// TIA Portal V19 export
FUNCTION "CallDiagnostic" : Void   // FC16, LAD
TITLE = Diagnostics / Diagnose
AUTHOR : Siemens Digital Industries
// Call of diagnostic blocks / Aufruf: Diagnose
// stored: IsIECCheckEnabled true, SetENOAutomatically true
   // Ret_Val : Ret_Val
BEGIN

REGION Network 1: Call Profinet Devices Diagnostics
   // For diagnostics of all profinet devices of this PLC
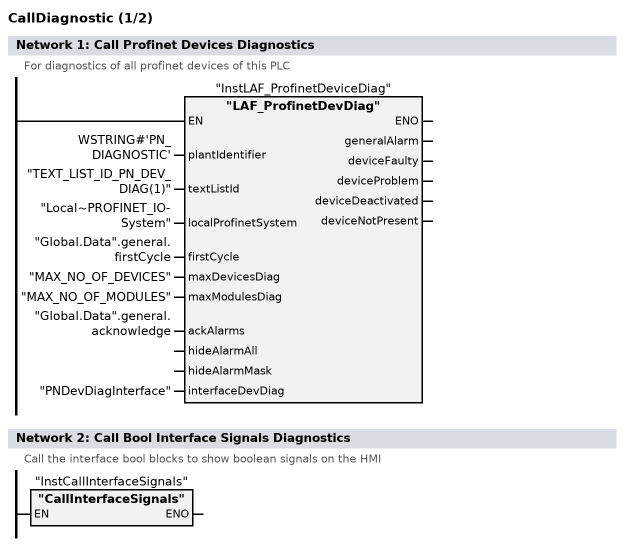
   RUNG wire#powerrail
      "InstLAF_ProfinetDeviceDiag"(plantIdentifier := WSTRING#'PN_DIAGNOSTIC', textListId := "TEXT_LIST_ID_PN_DEV_DIAG(1)", localProfinetSystem := "Local~PROFINET_IO-System", firstCycle := "Global.Data".general.firstCycle, maxDevicesDiag := "MAX_NO_OF_DEVICES", maxModulesDiag := "MAX_NO_OF_MODULES", ackAlarms := "Global.Data".general.acknowledge, hideAlarmAll :=, hideAlarmMask :=, interfaceDevDiag := "PNDevDiagInterface", generalAlarm =>, deviceFaulty =>, deviceProblem =>, deviceDeactivated =>, deviceNotPresent =>)
   END_RUNG
   // the same network as SCL:
   "InstLAF_ProfinetDeviceDiag"(plantIdentifier := WSTRING#'PN_DIAGNOSTIC',   // "LAF_ProfinetDevDiag"
                           textListId := "TEXT_LIST_ID_PN_DEV_DIAG(1)",
                           localProfinetSystem := "Local~PROFINET_IO-System",
                           firstCycle := "Global.Data".general.firstCycle,
                           maxDevicesDiag := "MAX_NO_OF_DEVICES",
                           maxModulesDiag := "MAX_NO_OF_MODULES",
                           ackAlarms := "Global.Data".general.acknowledge,
                           interfaceDevDiag := "PNDevDiagInterface");
END_REGION

REGION Network 2: Call Bool Interface Signals Diagnostics
   // Call the interface bool blocks to show boolean signals on the HMI
   RUNG wire#powerrail
      "InstCallInterfaceSignals"()
   END_RUNG
   // the same network as SCL:
   "InstCallInterfaceSignals"();   // "CallInterfaceSignals"
END_REGION

REGION Network 3: Call Drives Diagnostics
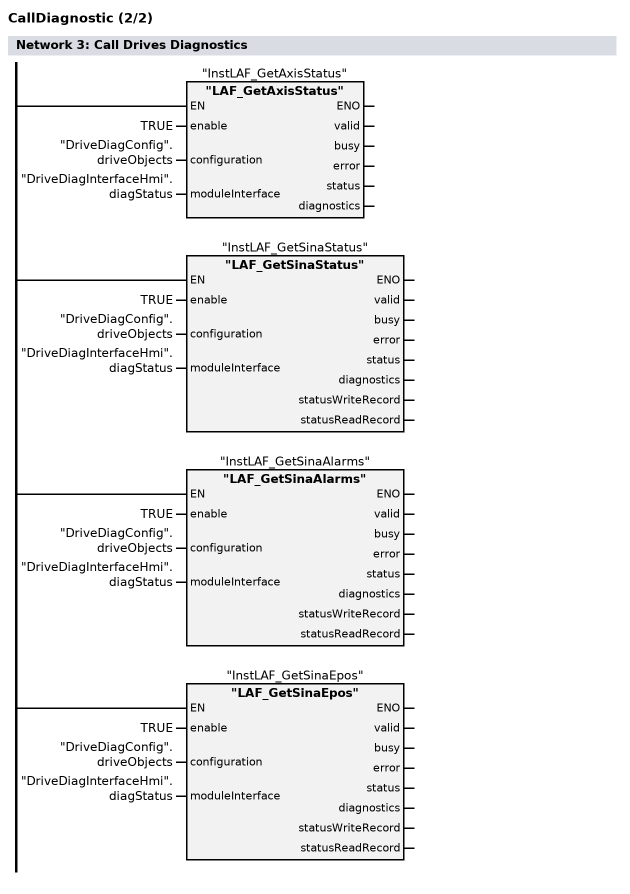
   RUNG wire#powerrail
      "InstLAF_GetAxisStatus"(enable := TRUE, configuration := "DriveDiagConfig".driveObjects, moduleInterface := "DriveDiagInterfaceHmi".diagStatus, valid =>, busy =>, error =>, status =>, diagnostics =>)
   END_RUNG
   RUNG wire#powerrail
      "InstLAF_GetSinaStatus"(enable := TRUE, configuration := "DriveDiagConfig".driveObjects, moduleInterface := "DriveDiagInterfaceHmi".diagStatus, valid =>, busy =>, error =>, status =>, diagnostics =>, statusWriteRecord =>, statusReadRecord =>)
   END_RUNG
   RUNG wire#powerrail
      "InstLAF_GetSinaAlarms"(enable := TRUE, configuration := "DriveDiagConfig".driveObjects, moduleInterface := "DriveDiagInterfaceHmi".diagStatus, valid =>, busy =>, error =>, status =>, diagnostics =>, statusWriteRecord =>, statusReadRecord =>)
   END_RUNG
   RUNG wire#powerrail
      "InstLAF_GetSinaEpos"(enable := TRUE, configuration := "DriveDiagConfig".driveObjects, moduleInterface := "DriveDiagInterfaceHmi".diagStatus, valid =>, busy =>, error =>, status =>, diagnostics =>, statusWriteRecord =>, statusReadRecord =>)
   END_RUNG
   // the same network as SCL:
   "InstLAF_GetAxisStatus"(enable := TRUE,   // "LAF_GetAxisStatus"
                           configuration := "DriveDiagConfig".driveObjects,
                           moduleInterface := "DriveDiagInterfaceHmi".diagStatus);
   "InstLAF_GetSinaStatus"(enable := TRUE,   // "LAF_GetSinaStatus"
                           configuration := "DriveDiagConfig".driveObjects,
                           moduleInterface := "DriveDiagInterfaceHmi".diagStatus);
   "InstLAF_GetSinaAlarms"(enable := TRUE,   // "LAF_GetSinaAlarms"
                           configuration := "DriveDiagConfig".driveObjects,
                           moduleInterface := "DriveDiagInterfaceHmi".diagStatus);
   "InstLAF_GetSinaEpos"(enable := TRUE,   // "LAF_GetSinaEpos"
                         configuration := "DriveDiagConfig".driveObjects,
                         moduleInterface := "DriveDiagInterfaceHmi".diagStatus);
END_REGION
END_FUNCTION
